TYPE SystemStatusWord :
STRUCT
	SysReady		:BOOL;		// System ist eingeschalten und bereit
	PrimReady		:BOOL;		// Primärreaktor ist bereit für den Prozess
	PrimActiv		:BOOL;		// Primärreaktor führt Prozess aus
	SekReady		:BOOL;		// Sekundärreaktor ist bereit für den Prozess
	SekActiv		:BOOL;		// Sekundärreaktor führt Prozess aus
	GF1Activ		:BOOL;		// Heiz- / Kühlprozess läuft
	GF2Activ		:BOOL;		// Entleerprozess läuft
	GF3Activ		:BOOL;		// Pumpprozess läuft
	GF4Activ		:BOOL;		// Halteprozess läuft
	GF5Activ		:BOOL;		// Rührprozess läuft
	GF6Activ		:BOOL;		// Warteprozess läuft
	GF7Activ		:BOOL;		// Auffüllprozess läuft
	GF8Activ		:BOOL;		// Zirkulierprozess läuft
END_STRUCT
END_TYPE

(* stored: Version 1.1.0.1, ProductVersion 3.1.4024.12
   DUT SystemStatusWord: Id {12b9cc79-7119-40fb-8a3d-043692b3e362} *)
